FUNCTION_BLOCK FB_MollineEHeatCounter
VAR_INPUT
	aHeatCounterTelegramm : ARRAY[1..cMBUS_MaxTelegrams] OF ST_MBus_Data2;
END_VAR
VAR_OUTPUT
	fFeedTemperature : REAL; //°C
	fReturnTemperature : REAL; //°C
	fVolumeFlowRate : REAL; //m3/h
	fHeatFlowRate : REAL; //kW
END_VAR
VAR
	{attribute 'OPC.UA.DA' := '1'}
	sensorState : ST_MollineC3HeatCounterState;
END_VAR

//set sensor state
sensorState.fVolume := STRING_TO_REAL(aHeatCounterTelegramm[1].arrData[3].sValue);
sensorState.fFeedTemperature := STRING_TO_REAL(aHeatCounterTelegramm[1].arrData[7].sValue);
sensorState.fReturnTemperature := STRING_TO_REAL(aHeatCounterTelegramm[1].arrData[8].sValue);
sensorState.fVolumeFlowRate := STRING_TO_REAL(aHeatCounterTelegramm[1].arrData[6].sValue);
sensorState.fHeatEnergy := STRING_TO_REAL(aHeatCounterTelegramm[1].arrData[2].sValue)/1000000;
sensorState.fTemperatureDifference := STRING_TO_REAL(aHeatCounterTelegramm[1].arrData[9].sValue);

//calculate fHeatFlowRate because heat meter does not measure negative flows
sensorState.fHeatFlowRate := sensorState.fVolumeFlowRate/3.6*4.19*sensorState.fTemperatureDifference;

//set outputs
fFeedTemperature := sensorState.fFeedTemperature;
fReturnTemperature := sensorState.fReturnTemperature;
fVolumeFlowRate := sensorState.fVolumeFlowRate;
fHeatFlowRate := sensorState.fHeatFlowRate;

END_FUNCTION_BLOCK

(* stored: Version 1.1.0.1, ProductVersion 3.1.4024.10
   POU FB_MollineEHeatCounter: Id {ef0baafb-281e-4df1-82a7-e1c83bf79f4b}, SpecialFunc None *)
